{attribute 'qualified_only'}
VAR_GLOBAL
    // 与外部Python Vision Service通过ADS交换的唯一螺钉角度视觉接口。
    stInterface : ST_ScrewVisionInterface;
END_VAR

(* stored: Version 1.1.0.1, ProductVersion 3.1.4026.20
   GVL GVL_ScrewVision: Id {448404D1-9E9A-48E5-9317-D0A441541D93} *)
